// TIA Portal V20 export
FUNCTION_BLOCK "FB_ExtLoadUnload"   // FB61, SCL
{ S7_Optimized_Access := 'TRUE' }
// stored: MemoryReserve 100, SetENOAutomatically false
   VAR_INPUT
      iStartSeqCond : Bool;   // Start Sequence Conditions
      iJobReq : Bool;   // Job Request - From Main
      iShuttleExtLoadUnloadAutoPos : Bool;   // Load/Unload Auto Pos. Reached - Param
      iShuttleExtLoadUnloadAutoPosSetPoint : LReal;   // Load/Unload Auto Pos. Setpoint - Param
      iShuttleExtLoadUnloadManuPos : Bool;   // Load/Unload Manu Pos. Reached - Param
      iShuttleExtLoadUnloadManuPosSetPoint : LReal;   // Load/Unload Manu Pos. Setpoint - Param
      iShuttleMoving : Bool;   // Shuttle is moving - From FB_LoaderAxis
      iShuttleInPos : Bool;   // Shuttle pos. reached - From FB_LoaderAxis
      iCommunicationWithExtLoaderDone : Bool;   // Communication Done - From Ext Loader
      iLoadUnloadMsgManuModeAck : Bool;   // Load/Unload Message Ack - From HMI
      iAutoMode : Bool;
      iSemiAutoMode : Bool;
      iFillingMode : Bool;   // Filling Mode - From Machine States
      iEmptyingMode : Bool;   // Emptying Mode - From Machine States
      iPLC_DateAndTime : DTL;
      iStepPause : Bool;
   END_VAR
   VAR_OUTPUT
      oShuttleStartReq { ExternalAccessible := 'False'; ExternalVisible := 'False'; ExternalWritable := 'False'} : Bool;   // Shuttle Start Order - To FB_LoaderAxis
      oShuttlePosSetPoint { ExternalAccessible := 'False'; ExternalVisible := 'False'; ExternalWritable := 'False'} : Real;   // Shuttle Position Setpoint - To FB_LoaderAxis
      oStartCommunicationWithExtLoader : Bool;   // Start Communication - To Ext Loader
      oSetLoadUnloadMsgManuMode : Bool;   // Set Load/Unload Message - To HMI
   END_VAR
   VAR
      sCurrent_Step_NB : Int;   // Active Step Number
      sCheck_Step_Condition : Bool;
      sOneStepForward : Bool;
      sRTOneStepForward : R_TRIG;
      sOneStepMode { S7_SetPoint := 'True'} : Bool;
      sStepForward : Bool;
      sInterface : "UDT_SequenceInterface";
      sShuttleStartReq { ExternalAccessible := 'False'; ExternalVisible := 'False'; ExternalWritable := 'False'} : Bool;
      sShuttlePosSetPoint { ExternalAccessible := 'False'; ExternalVisible := 'False'; ExternalWritable := 'False'} : Real;
      sHistory : Struct
         Activation : Bool;
         Steps : Array[0..99] of Int;
         Date_Time : Array[0..99] of DTL;
      END_STRUCT;
      StepText : "FB_GetTextErrorCode";
   END_VAR
   VAR_TEMP
      tIndex : Int;   // Index
   END_VAR
   VAR CONSTANT
      S00_INIT : Int := 0;
      S10_CHECK_EXT_LOAD_UNLOAD_OPTION : Int := 10;
      S20_SHUTTLE_TO_EXT_LOAD_UNLOAD_POS_START_REQ : Int := 20;
      S30_SHUTTLE_TO_EXT_LOAD_UNLOAD_POS_REACHED : Int := 30;
      S40_SET_EXCHANGE_EXT_LOADER_LOAD_UNLOAD : Int := 40;
      S50_EXCHANGE_EXT_LOADER_IN_PROGRESS : Int := 50;
      S60_EXCHANGE_EXT_LOADER_ACQUIT : Int := 60;
      S70_SET_EXCHANGE_EXT_LOADER_UNLOAD : Int := 70;
      S80_EXCHANGE_EXT_LOADER_IN_PROGRESS : Int := 80;
      S90_EXCHANGE_EXT_LOADER_ACQUIT : Int := 90;
      S100_SET_EXCHANGE_EXT_LOADER_UNLOAD : Int := 100;
      S110_EXCHANGE_EXT_LOADER_IN_PROGRESS : Int := 110;
      S120_EXCHANGE_EXT_LOADER_ACQUIT : Int := 120;
      S130_SHUTTLE_TO_EXT_LOAD_UNLOAD_MANU_POS_START_REQ : Int := 130;
      S140_SHUTTLE_TO_EXT_LOAD_UNLOAD_MANU_POS_REACHED : Int := 140;
      S150_OPERATOR_MESSAGE : Int := 150;
      S195_JOB_DONE : Int := 195;
   END_VAR
   // StepText.sCode_error[0].ErrorCode := 0;
   // StepText.sCode_error[1].ErrorCode := 10;
   // StepText.sCode_error[2].ErrorCode := 20;
   // StepText.sCode_error[3].ErrorCode := 30;
   // StepText.sCode_error[4].ErrorCode := 40;
   // StepText.sCode_error[5].ErrorCode := 50;
   // StepText.sCode_error[6].ErrorCode := 60;
   // StepText.sCode_error[7].ErrorCode := 70;
   // StepText.sCode_error[8].ErrorCode := 80;
   // StepText.sCode_error[9].ErrorCode := 90;
   // StepText.sCode_error[10].ErrorCode := 95;
BEGIN
   REGION Description header 
       //==================================================================================
       // POSALUX Swiss SA / (C) Copyright 2025
       //----------------------------------------------------------------------------------
       // Title: FB_ExtLoadUnload
       // Comment/Function: 
       // Author: Fabien WALDT
       // Engineering: TIA Portal v17
       //----------------------------------------------------------------------------------
       // Change log table:
       // Version  | Date     | Expert in charge | Changes applied
       // ---------|----------|------------------|-----------------------------------------
       // 00.00.01 | 20250527 | WFA              | First released version
       // =================================================================================
   END_REGION

   REGION Define condition to start
       IF #iStartSeqCond THEN
           #sInterface.SequenceReleased := TRUE;
       ELSE
           // Standard sequencer controls
           #sInterface.SequenceReleased := FALSE;
           #sCurrent_Step_NB := #S00_INIT;
           #sInterface.SequenceRun := FALSE;
           #sInterface.JobDone := FALSE;
           #sCheck_Step_Condition := FALSE;

           // Dedicated sequencer controls
           #sShuttleStartReq := FALSE;
           #sShuttlePosSetPoint := 0.0;
           #oStartCommunicationWithExtLoader := FALSE;
           // Add specifics controls 
       END_IF;

       // Reset interface error
       IF #sInterface.Reset THEN
           #sInterface.Error := FALSE;
       END_IF;

       // Reset start when axis in position
       IF #iShuttleInPos THEN
           #sShuttleStartReq := FALSE;
       END_IF;

       // One step forward
       #sRTOneStepForward.CLK := #sOneStepForward;
       #sRTOneStepForward();
       #sStepForward := (NOT #sOneStepMode OR (#sOneStepMode AND #sRTOneStepForward.Q)) AND NOT #iStepPause;
       #sOneStepForward := FALSE;

       // Action only true in dedicated steps
       #oSetLoadUnloadMsgManuMode := FALSE;
   END_REGION

   REGION Sequence Function
       CASE #sCurrent_Step_NB OF
           #S00_INIT:
               REGION S00 INIT
                   #sCheck_Step_Condition := TRUE;
               END_REGION
           #S10_CHECK_EXT_LOAD_UNLOAD_OPTION:
               REGION S10_CHECK_EXT_LOAD_UNLOAD_OPTION
                   #sCheck_Step_Condition := TRUE;
               END_REGION
           #S20_SHUTTLE_TO_EXT_LOAD_UNLOAD_POS_START_REQ:
               REGION S20_SHUTTLE_TO_EXT_LOAD_UNLOAD_POS_START_REQ
                   #sShuttleStartReq := NOT #iShuttleExtLoadUnloadAutoPos;
                   #sShuttlePosSetPoint := LREAL_TO_REAL(#iShuttleExtLoadUnloadAutoPosSetPoint);
                   #sCheck_Step_Condition := TRUE;
               END_REGION
           #S30_SHUTTLE_TO_EXT_LOAD_UNLOAD_POS_REACHED:
               REGION S30_SHUTTLE_TO_EXT_LOAD_UNLOAD_POS_REACHED
                   #sCheck_Step_Condition := TRUE;
               END_REGION
           #S40_SET_EXCHANGE_EXT_LOADER_LOAD_UNLOAD:
               REGION S40_SET_EXCHANGE_EXT_LOADER_LOAD_UNLOAD
                   #oStartCommunicationWithExtLoader := TRUE;
                   #sCheck_Step_Condition := TRUE;
               END_REGION
           #S50_EXCHANGE_EXT_LOADER_IN_PROGRESS:
               REGION S50_EXCHANGE_EXT_LOADER_IN_PROGRESS
                   #sCheck_Step_Condition := TRUE;
               END_REGION
           #S60_EXCHANGE_EXT_LOADER_ACQUIT:
               REGION S60_EXCHANGE_EXT_LOADER_ACQUIT
                   #oStartCommunicationWithExtLoader := FALSE;
                   #sCheck_Step_Condition := TRUE;
               END_REGION
           #S70_SET_EXCHANGE_EXT_LOADER_UNLOAD:
               REGION S70_SET_EXCHANGE_EXT_LOADER_UNLOAD
                   #oStartCommunicationWithExtLoader := TRUE;
                   #sCheck_Step_Condition := TRUE;
               END_REGION
           #S80_EXCHANGE_EXT_LOADER_IN_PROGRESS:
               REGION S80_EXCHANGE_EXT_LOADER_IN_PROGRESS
                   #sCheck_Step_Condition := TRUE;
               END_REGION
           #S90_EXCHANGE_EXT_LOADER_ACQUIT:
               REGION S90_EXCHANGE_EXT_LOADER_ACQUIT
                   #oStartCommunicationWithExtLoader := FALSE;
                   #sCheck_Step_Condition := TRUE;
               END_REGION
           #S100_SET_EXCHANGE_EXT_LOADER_UNLOAD:
               REGION S100_SET_EXCHANGE_EXT_LOADER_UNLOAD
                   #oStartCommunicationWithExtLoader := TRUE;
                   #sCheck_Step_Condition := TRUE;
               END_REGION
           #S110_EXCHANGE_EXT_LOADER_IN_PROGRESS:
               REGION S110_EXCHANGE_EXT_LOADER_IN_PROGRESS
                   #sCheck_Step_Condition := TRUE;
               END_REGION
           #S120_EXCHANGE_EXT_LOADER_ACQUIT:
               REGION S120_EXCHANGE_EXT_LOADER_ACQUIT
                   #oStartCommunicationWithExtLoader := FALSE;
                   #sCheck_Step_Condition := TRUE;
               END_REGION
           #S130_SHUTTLE_TO_EXT_LOAD_UNLOAD_MANU_POS_START_REQ:
               REGION S130_SHUTTLE_TO_EXT_LOAD_UNLOAD_MANU_POS_START_REQ
                   #sShuttleStartReq := NOT #iShuttleExtLoadUnloadManuPos;
                   #sShuttlePosSetPoint := LREAL_TO_REAL(#iShuttleExtLoadUnloadManuPosSetPoint);
                   #sCheck_Step_Condition := TRUE;
               END_REGION
           #S140_SHUTTLE_TO_EXT_LOAD_UNLOAD_MANU_POS_REACHED:
               REGION S140_SHUTTLE_TO_EXT_LOAD_UNLOAD_MANU_POS_REACHED
                   #sCheck_Step_Condition := TRUE;
               END_REGION
           #S150_OPERATOR_MESSAGE:
               REGION S150_OPERATOR_MESSAGE
                   #oSetLoadUnloadMsgManuMode := TRUE;
                   #sCheck_Step_Condition := TRUE;
               END_REGION
           #S195_JOB_DONE:
               REGION S95_JOB_DONE
                   #sInterface.JobDone := TRUE;
                   #sCheck_Step_Condition := TRUE;
               END_REGION
           ELSE:
               #sInterface.Error := TRUE;
       END_CASE;
   END_REGION

   REGION Sequence Next Step Condition
       IF #sCheck_Step_Condition THEN
           CASE #sCurrent_Step_NB OF
               #S00_INIT:
                   REGION S00 INIT
                       IF #sInterface.SequenceReleased AND #iJobReq THEN
                           #sCurrent_Step_NB := #S10_CHECK_EXT_LOAD_UNLOAD_OPTION;
                           #sInterface.SequenceRun := TRUE;
                           #sCheck_Step_Condition := FALSE;
                       ELSE
                           #sInterface.SequenceRun := FALSE;
                       END_IF;
                   END_REGION
               #S10_CHECK_EXT_LOAD_UNLOAD_OPTION:
                   REGION S10_CHECK_EXT_LOAD_UNLOAD_OPTION
                       IF #sInterface.SequenceReleased AND #sStepForward AND "DB_LoaderOptions".ExtLoadUnload.CommonPos AND #iAutoMode THEN
                           #sCurrent_Step_NB := #S20_SHUTTLE_TO_EXT_LOAD_UNLOAD_POS_START_REQ;
                           #sCheck_Step_Condition := FALSE;
                       ELSIF #sInterface.SequenceReleased AND #sStepForward AND #iSemiAutoMode THEN
                           #sCurrent_Step_NB := #S130_SHUTTLE_TO_EXT_LOAD_UNLOAD_MANU_POS_START_REQ;
                           #sCheck_Step_Condition := FALSE;
                       END_IF;
                   END_REGION
               #S20_SHUTTLE_TO_EXT_LOAD_UNLOAD_POS_START_REQ:
                   REGION S20_SHUTTLE_TO_EXT_LOAD_UNLOAD_POS_START_REQ
                       IF #sInterface.SequenceReleased AND (#iShuttleMoving OR #iShuttleExtLoadUnloadAutoPos) THEN
                           #sCurrent_Step_NB := #S30_SHUTTLE_TO_EXT_LOAD_UNLOAD_POS_REACHED;
                           #sCheck_Step_Condition := FALSE;
                       END_IF;
                   END_REGION
               #S30_SHUTTLE_TO_EXT_LOAD_UNLOAD_POS_REACHED:
                   REGION S30_SHUTTLE_TO_EXT_LOAD_UNLOAD_POS_REACHED
                       IF #sInterface.SequenceReleased AND #sStepForward AND NOT #sShuttleStartReq AND #iShuttleExtLoadUnloadAutoPos AND NOT #iEmptyingMode AND NOT #iFillingMode THEN
                           #sCurrent_Step_NB := #S40_SET_EXCHANGE_EXT_LOADER_LOAD_UNLOAD;
                           #sCheck_Step_Condition := FALSE;
                       ELSIF #sInterface.SequenceReleased AND #sStepForward AND NOT #sShuttleStartReq AND #iShuttleExtLoadUnloadAutoPos AND #iEmptyingMode AND NOT #iFillingMode THEN
                           #sCurrent_Step_NB := #S70_SET_EXCHANGE_EXT_LOADER_UNLOAD;
                           #sCheck_Step_Condition := FALSE;
                       ELSIF #sInterface.SequenceReleased AND #sStepForward AND NOT #sShuttleStartReq AND #iShuttleExtLoadUnloadAutoPos AND NOT #iEmptyingMode AND #iFillingMode THEN
                           #sCurrent_Step_NB := #S100_SET_EXCHANGE_EXT_LOADER_UNLOAD;
                           #sCheck_Step_Condition := FALSE;
                       END_IF;
                   END_REGION
               #S40_SET_EXCHANGE_EXT_LOADER_LOAD_UNLOAD:
                   REGION S40_SET_EXCHANGE_EXT_LOADER_LOAD_UNLOAD
                       IF #sInterface.SequenceReleased AND #sStepForward AND "AlwaysTRUE" THEN
                           #sCurrent_Step_NB := #S50_EXCHANGE_EXT_LOADER_IN_PROGRESS;
                           #sCheck_Step_Condition := FALSE;
                       END_IF;
                   END_REGION
               #S50_EXCHANGE_EXT_LOADER_IN_PROGRESS:
                   REGION S50_EXCHANGE_EXT_LOADER_IN_PROGRESS
                       IF #sInterface.SequenceReleased AND #sStepForward AND #iCommunicationWithExtLoaderDone THEN
                           #sCurrent_Step_NB := #S60_EXCHANGE_EXT_LOADER_ACQUIT;
                           #sCheck_Step_Condition := FALSE;
                       END_IF;
                   END_REGION
               #S60_EXCHANGE_EXT_LOADER_ACQUIT:
                   REGION S60_EXCHANGE_EXT_LOADER_ACQUIT
                       IF #sInterface.SequenceReleased AND #sStepForward AND "AlwaysTRUE" THEN
                           #sCurrent_Step_NB := #S195_JOB_DONE;
                           #sCheck_Step_Condition := FALSE;
                       END_IF;
                   END_REGION
               #S70_SET_EXCHANGE_EXT_LOADER_UNLOAD:
                   REGION S70_SET_EXCHANGE_EXT_LOADER_UNLOAD
                       IF #sInterface.SequenceReleased AND #sStepForward AND "AlwaysTRUE" THEN
                           #sCurrent_Step_NB := #S80_EXCHANGE_EXT_LOADER_IN_PROGRESS;
                           #sCheck_Step_Condition := FALSE;
                       END_IF;
                   END_REGION
               #S80_EXCHANGE_EXT_LOADER_IN_PROGRESS:
                   REGION S80_EXCHANGE_EXT_LOADER_IN_PROGRESS
                       IF #sInterface.SequenceReleased AND #sStepForward AND #iCommunicationWithExtLoaderDone THEN
                           #sCurrent_Step_NB := #S90_EXCHANGE_EXT_LOADER_ACQUIT;
                           #sCheck_Step_Condition := FALSE;
                       END_IF;
                   END_REGION
               #S90_EXCHANGE_EXT_LOADER_ACQUIT:
                   REGION S90_EXCHANGE_EXT_LOADER_ACQUIT
                       IF #sInterface.SequenceReleased AND #sStepForward AND "AlwaysTRUE" THEN
                           #sCurrent_Step_NB := #S195_JOB_DONE;
                           #sCheck_Step_Condition := FALSE;
                       END_IF;
                   END_REGION
               #S100_SET_EXCHANGE_EXT_LOADER_UNLOAD:
                   REGION S100_SET_EXCHANGE_EXT_LOADER_UNLOAD
                       IF #sInterface.SequenceReleased AND #sStepForward AND "AlwaysTRUE" THEN
                           #sCurrent_Step_NB := #S110_EXCHANGE_EXT_LOADER_IN_PROGRESS;
                           #sCheck_Step_Condition := FALSE;
                       END_IF;
                   END_REGION
               #S110_EXCHANGE_EXT_LOADER_IN_PROGRESS:
                   REGION S110_EXCHANGE_EXT_LOADER_IN_PROGRESS
                       IF #sInterface.SequenceReleased AND #sStepForward AND #iCommunicationWithExtLoaderDone THEN
                           #sCurrent_Step_NB := #S120_EXCHANGE_EXT_LOADER_ACQUIT;
                           #sCheck_Step_Condition := FALSE;
                       END_IF;
                   END_REGION
               #S120_EXCHANGE_EXT_LOADER_ACQUIT:
                   REGION S120_EXCHANGE_EXT_LOADER_ACQUIT
                       IF #sInterface.SequenceReleased AND #sStepForward AND "AlwaysTRUE" THEN
                           #sCurrent_Step_NB := #S195_JOB_DONE;
                           #sCheck_Step_Condition := FALSE;
                       END_IF;
                   END_REGION
               #S130_SHUTTLE_TO_EXT_LOAD_UNLOAD_MANU_POS_START_REQ:
                   REGION S130_SHUTTLE_TO_EXT_LOAD_UNLOAD_MANU_POS_START_REQ
                       IF #sInterface.SequenceReleased AND (#iShuttleMoving OR #iShuttleExtLoadUnloadManuPos) THEN
                           #sCurrent_Step_NB := #S140_SHUTTLE_TO_EXT_LOAD_UNLOAD_MANU_POS_REACHED;
                           #sCheck_Step_Condition := FALSE;
                       END_IF;
                   END_REGION
               #S140_SHUTTLE_TO_EXT_LOAD_UNLOAD_MANU_POS_REACHED:
                   REGION S140_SHUTTLE_TO_EXT_LOAD_UNLOAD_MANU_POS_REACHED
                       IF #sInterface.SequenceReleased AND #sStepForward AND NOT #sShuttleStartReq AND #iShuttleExtLoadUnloadManuPos THEN
                           #sCurrent_Step_NB := #S150_OPERATOR_MESSAGE;
                           #sCheck_Step_Condition := FALSE;
                       END_IF;
                   END_REGION
               #S150_OPERATOR_MESSAGE:
                   REGION S150_OPERATOR_MESSAGE
                       IF #sInterface.SequenceReleased AND #sStepForward AND #iLoadUnloadMsgManuModeAck THEN
                           #sCurrent_Step_NB := #S195_JOB_DONE;
                           #sCheck_Step_Condition := FALSE;
                       END_IF;
                   END_REGION
               #S195_JOB_DONE:
                   REGION S95_JOB_DONE
                       IF NOT #iJobReq THEN
                           #sCurrent_Step_NB := #S00_INIT;
                           #sCheck_Step_Condition := FALSE;
                           #sInterface.JobDone := FALSE;
                       END_IF;
                   END_REGION
               ELSE
                   #sInterface.Error := TRUE;
           END_CASE;
       END_IF;
   END_REGION

   REGION Outputs Update
       #oShuttleStartReq := #sShuttleStartReq;
       #oShuttlePosSetPoint := #sShuttlePosSetPoint;
   END_REGION

   REGION Steps - Date and Time History
       IF #sHistory.Activation THEN
           IF #sHistory.Steps[0] <> #sCurrent_Step_NB THEN
               FOR #tIndex := 98 TO 0 BY -1 DO
                   #sHistory.Steps[#tIndex + 1] := #sHistory.Steps[#tIndex];
                   #sHistory.Date_Time[#tIndex + 1] := #sHistory.Date_Time[#tIndex];
               END_FOR;
               #sHistory.Steps[0] := #sCurrent_Step_NB;
               #sHistory.Date_Time[0] := #iPLC_DateAndTime;
           END_IF;
       END_IF;
   END_REGION

   REGION Steps Text
       #StepText(iErrorCode := #sCurrent_Step_NB,
                 oErrorText => #StepText.oErrorText);
   END_REGION
END_FUNCTION_BLOCK
